{attribute 'qualified_only'}
VAR_GLOBAL
END_VAR

(* stored: Version 1.1.0.1, ProductVersion 3.1.4024.12
   GVL GVL_Data: Id {d8a9d773-1adb-4903-b2fd-997e2b005b6e} *)
